// 隐含生成代码：不要编辑
FUNCTION CheckDivReal : REAL
VAR_INPUT
	divisor:REAL;
END_VAR

// 隐含生成代码：这里只是对代码实现的建议
{noflow}
IF divisor = 0 THEN
	CheckDivReal:=1;
ELSE
	CheckDivReal:=divisor;
END_IF;
{flow}

END_FUNCTION

(* stored: Version 1.1.0.1, ProductVersion 3.1.4024.9
   POU CheckDivReal: Id {80de408c-79d9-4fd8-9f9b-43c53f5ba82a}, SpecialFunc CheckDivReal32 *)
